// LS Electric XG5000 project: 타이머 3개
// PLC NewPLC

PROGRAM NewProgram (task: 스캔 프로그램)

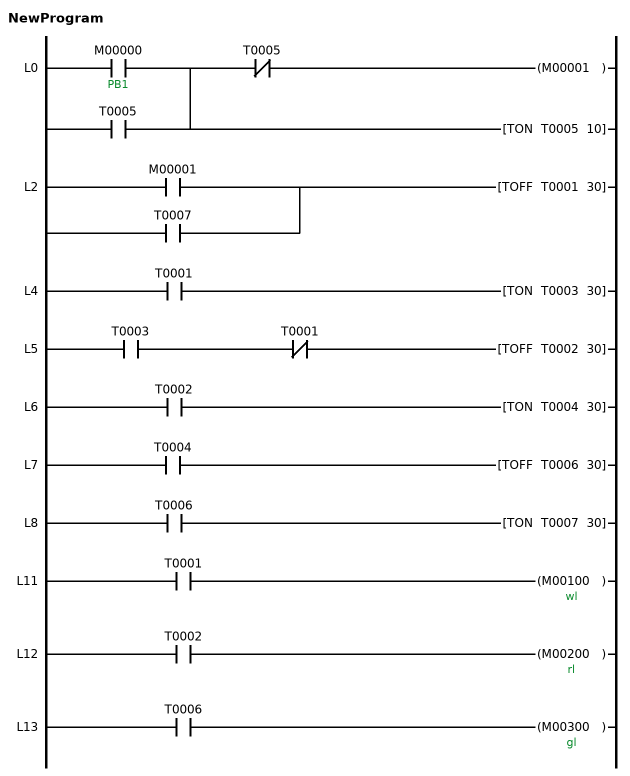
; L0
LOAD      M00000	// PB1
OR        T0005
MPUSH
AND NOT   T0005
OUT       M00001
MPOP
TON       T0005 10
; L2
LOAD      M00001
OR        T0007
TOFF      T0001 30
; L4
LOAD      T0001
TON       T0003 30
; L5
LOAD      T0003
AND NOT   T0001
TOFF      T0002 30
; L6
LOAD      T0002
TON       T0004 30
; L7
LOAD      T0004
TOFF      T0006 30
; L8
LOAD      T0006
TON       T0007 30
; L11
LOAD      T0001
OUT       M00100	// wl
; L12
LOAD      T0002
OUT       M00200	// rl
; L13
LOAD      T0006
OUT       M00300	// gl